INTERFACE I_Node EXTENDS I_NodePrototype, I_Disposable, I_HostContent, I_HostInputPorts, I_HostOutputPorts, I_HostAlarms, I_HostParameters, I_HostExtensions, I_HostMetadata, I_EventEmitter, I_Deserializable, I_Serializable

METHOD PUBLIC Accept
VAR_INPUT
	Visitor : I_NodeVisitor;
END_VAR
END_METHOD

METHOD PUBLIC Execute
END_METHOD

PROPERTY PUBLIC Id : T_MAXSTRING
GET
END_GET
END_PROPERTY

PROPERTY PUBLIC Mode : DINT
GET
END_GET
END_PROPERTY

PROPERTY PUBLIC Order : DINT
GET
END_GET
END_PROPERTY

END_INTERFACE

(* stored: Version 1.1.0.1, ProductVersion 3.1.4024.12
   Itf I_Node: Id {7e28b21d-6b2a-0b88-18bc-3ad32fd1a6c2}
   Method Accept: Id {9a7ac280-4430-0727-2fa0-fc419b9e7a74}
   Method Execute: Id {7f9f5b88-6b3e-01b0-3c44-302ecbab1d70}
   Property Id: Id {3f0a605f-e0ca-0b68-32ae-dc045045cbef}
   Get Get: Id {9693ab0f-432b-03b3-2695-d2bcd82c6f64}
   Property Mode: Id {ec3476cc-9f6e-0390-3d95-a2e1e0263e0e}
   Get Get: Id {d5d5fc57-033b-053e-0bee-8afed9f6afe1}
   Property Order: Id {7def7f08-10ff-0b9f-31cc-0ffdbdb8a639}
   Get Get: Id {e8fce107-543d-02d8-0594-172e06e8a866} *)
